FUNCTION Convert_USINT_TO_SINT : Hresult
VAR_INPUT
	in : USINT;
	out : REFERENCE TO SINT;
END_VAR
VAR
	converted : SINT;
END_VAR
VAR CONSTANT
	INCOMPATIBLE : HRESULT := 16#9811070E;
END_VAR

converted := USINT_TO_SINT(in);

IF (SINT_TO_USINT(converted) <> in) THEN
	Convert_USINT_TO_SINT := INCOMPATIBLE;
	RETURN;
END_IF

out := converted;

END_FUNCTION

(* stored: Version 1.1.0.1, ProductVersion 3.1.4024.12
   POU Convert_USINT_TO_SINT: Id {d7ded20e-f75c-4eaa-99c8-836461836115}, SpecialFunc None *)
